PROGRAM MAIN
VAR
END_VAR

P_EventsSimple();

END_PROGRAM

(* stored: Version 1.1.0.1, ProductVersion 3.1.4024.3
   POU MAIN: Id {6cd17c2e-3b65-472b-983b-233e74757831}, SpecialFunc None *)
